INTERFACE I_ToString EXTENDS I_Base

METHOD ToString : T_MaxString
VAR_INPUT
END_VAR
END_METHOD

END_INTERFACE

(* stored: Version 1.1.0.1
   Itf I_ToString: Id {0c57047e-fe76-4078-a8ef-709bfe3aa1b6}
   Method ToString: Id {24019f64-abfe-40cc-9e5d-fe93e3ac8762} *)
